TYPE RADII_LIMIT :
STRUCT
    LOW_LIMIT  : REAL := 0;     //Lowest allowed radius
    HIGH_LIMIT : REAL := 10000; //Highest allowed radius
END_STRUCT
END_TYPE

(* stored: Version 1.1.0.1, ProductVersion 3.1.4020.12
   DUT RADII_LIMIT: Id {c1816cb3-ac1b-4d82-848e-a830039fe351} *)
